(* IEC 61131-3 sources: CodesysTest/export/SX.dev/Plc Logic/Application, 8 files *)

(* ---- Counters.gvl.st ---- *)
(*#-#-#-#-#-#-#-#-#-#---Declaration---#-#-#-#-#-#-#-#-#-#-#-#-#*)

{attribute 'qualified_only'}
VAR_GLOBAL
	jawCycleTestCount : FB_MachineCounter(name := 'Jaw Cycle Test Counter');
	baggerCycles : FB_MachineCounter(name := 'Bagger Cycle Counter');
	pressureBarCycles : FB_MachineCounter(name := 'Pressure Bar Cycle Counter');
	(*Counters*)

	//passthroughChanges : FB_MachineCounter(name := 'Passthrough Changes Counter');
	//loadPlateCycles : FB_MachineCounter(name := 'Load Plate Cycle Counter');
	//printerCycles : FB_MachineCounter(name := 'Printer Cycle Counter');
	//motorizedSealFlattenerCycles : FB_MachineCounter(name := 'Motorized Seal Flattener Cycles');
	//bagOpenRetryTotal : FB_MachineCounter(name := 'Bag Open Retry Totals');
END_VAR

(* ---- Globals.gvl.st ---- *)
(*#-#-#-#-#-#-#-#-#-#---Declaration---#-#-#-#-#-#-#-#-#-#-#-#-#*)

{attribute 'qualified_only'}
{attribute 'global_init_slot' := '49994'}
VAR_GLOBAL
	SystemLog : FB_InternalLogger;

END_VAR

VAR_GLOBAL CONSTANT
	MAX_LOGGED_ITEMS : UINT := 500;	// Max items to be logged
	STEPS_PER_INCH_IBD : DINT := 1250;
	STEPS_PER_INCH_JAW : DINT := 1250;
	STEPS_PER_INCH_LOAD_PLATE : DINT := 931;
	STEPS_PER_INCH_FILM : DINT := 1000;
	SERIAL_BUFFER_SIZE : BYTE := 50;
	SEAL_TO_PHOTOEYE_DISTANCE : REAL := 4.65;
END_VAR

(* ---- PersistentVars.gvl.st ---- *)
(*#-#-#-#-#-#-#-#-#-#---Declaration---#-#-#-#-#-#-#-#-#-#-#-#-#*)

{attribute 'qualified_only'}
VAR_GLOBAL PERSISTENT RETAIN
	// Generated instance path of persistent variable
	HMIData.bagsMade: UDINT;
	// Generated instance path of persistent variable
	HMIData.batchEnable: BOOL;
	// Generated instance path of persistent variable
	HMIData.batchSetting: UDINT := UDINT#10;
	// Generated instance path of persistent variable
	HMIData.batchCount: UDINT;
	// Generated instance path of persistent variable
	HMIData.headCycleCount: UDINT;
	// Generated instance path of persistent variable
	HMIData.pressureBarOpenDelay: REAL;
	// Generated instance path of persistent variable
	HMIData.pressureBarCloseDelay: REAL;
	// Generated instance path of persistent variable
	HMIData.passthroughSetting: REAL := REAL#5.5;
	// Generated instance path of persistent variable
	HMIData.sealBarDwell: REAL := REAL#0.18;
	// Generated instance path of persistent variable
	HMIData.sealBarCool: REAL := REAL#0.25;
	// Generated instance path of persistent variable
	HMIData.bagSkirtLength: REAL := 2.0;
	// Generated instance path of persistent variable
	HMIData.bagLength: REAL := REAL#17.62;
	// Generated instance path of persistent variable
	HMIData.bagWidth: REAL := 11.0;
	// Generated instance path of persistent variable
	HMIData.bagThickness: REAL := REAL#2.5;
	// Generated instance path of persistent variable
	HMIData.bagForwardSpeed: UDINT := UDINT#40;
	// Generated instance path of persistent variable
	HMIData.bagReverseSpeed: UDINT := UDINT#8;
	// Generated instance path of persistent variable
	HMIData.printSpeed: UDINT := UDINT#6;
	// Generated instance path of persistent variable
	HMIData.printLength: REAL := REAL#3;
	// Generated instance path of persistent variable
	HMIData.printOffset: REAL := REAL#8;
	// Generated instance path of persistent variable
	HMIData.fillerCountSetting: UDINT;
	// Generated instance path of persistent variable
	HMIData.fillerCurrentCount: UDINT;
	// Generated instance path of persistent variable
	HMIData.fillerDropTime: REAL;
	// Generated instance path of persistent variable
	HMIData.loadPlateDelay: REAL;
	// Generated instance path of persistent variable
	HMIData.loadPlateDwell: REAL := REAL#0.1;
	// Generated instance path of persistent variable
	HMIData.IBDInUse: BOOL := TRUE;
	// Generated instance path of persistent variable
	HMIData.IBDInstalled: BOOL := TRUE;
	// Generated instance path of persistent variable
	HMIData.IBDOpenMotionProfile: sctMotionProfile := STRUCT(velo := REAL#9, accel := REAL#30, decel := REAL#50, current := REAL#100);
	// Generated instance path of persistent variable
	HMIData.IBDCloseMotionProfile: sctMotionProfile := STRUCT(velo := REAL#15, accel := REAL#10, decel := REAL#10, current := REAL#50);
	// Generated instance path of persistent variable
	HMIData.IBDZeroOffset: REAL := REAL#2;
	// Generated instance path of persistent variable
	HMIData.jawCloseDelay: REAL := REAL#0.1;
	// Generated instance path of persistent variable
	HMIData.jawClosePositionSetting: REAL := REAL#-0.45;
	// Generated instance path of persistent variable
	HMIData.jawOpenMotionProfile: sctMotionProfile := STRUCT(velo := REAL#14, accel := REAL#300, decel := REAL#300, current := REAL#100);
	// Generated instance path of persistent variable
	HMIData.jawCloseMotionProfile: sctMotionProfile := STRUCT(velo := REAL#14, accel := REAL#10, decel := REAL#10, current := REAL#100);
	// Generated instance path of persistent variable
	HMIData.jawCycleTestCycles: DINT;
	// Generated instance path of persistent variable
	HMIData.jawCycleTestActive: BOOL;
	// Generated instance path of persistent variable
	HMIData.jawZeroOffset: REAL := REAL#2;
	// Generated instance path of persistent variable
	HMIData.lastCycleTime: REAL;
	// Generated instance path of persistent variable
	HMIData.bagDropClearanceDwell: REAL := REAL#0.5;
	// Generated instance path of persistent variable
	HMIData.averageCycleTime: REAL;
	// Generated instance path of persistent variable
	HMIData.currentJobID: INT;
	// Generated instance path of persistent variable
	HMIData.separateBeforeSeal: BOOL := TRUE;
	// Generated instance path of persistent variable
	HMIData.partsCounterEnable: BOOL;
	// Generated instance path of persistent variable
	HMIData.partsCounterCount: UDINT;
	// Generated instance path of persistent variable
	HMIData.partsCounterSetting: UDINT;
	// Generated instance path of persistent variable
	HMIData.consecutiveBagsEnable: BOOL;
	// Generated instance path of persistent variable
	HMIData.consecutiveBagsCount: UDINT;
	// Generated instance path of persistent variable
	HMIData.consecutiveBagsSetting: UDINT;
	// Generated instance path of persistent variable
	HMIData.printerInstalled: BOOL := TRUE;
	// Generated instance path of persistent variable
	HMIData.printerInUse: BOOL := TRUE;
	// Generated instance path of persistent variable
	HMIData.printerCancelRequest: BOOL;
	// Generated instance path of persistent variable
	HMIData.barcodeVerifierInstalled: BOOL := TRUE;
	// Generated instance path of persistent variable
	HMIData.barcodeGoodReadCount: UDINT;
	// Generated instance path of persistent variable
	HMIData.barcodeBadReadCount: UDINT;
	// Generated instance path of persistent variable
	HMIData.barcodeBadReadFaultSetting: UDINT;
	// Generated instance path of persistent variable
	HMIData.barcodeStartPosition: REAL;
	// Generated instance path of persistent variable
	HMIData.barcodeScanDistance: REAL := REAL#1;
	// Generated instance path of persistent variable
	HMIData.barcodeVerifierInUse: BOOL := TRUE;
	// Generated instance path of persistent variable
	HMIData.loadPlateInstalled: BOOL := TRUE;
	// Generated instance path of persistent variable
	HMIData.loadPlateLoweredPositionSetting: REAL := 0.0;
	// Generated instance path of persistent variable
	HMIData.loadPlateRaisedPositionSetting: REAL := 1.0;
	// Generated instance path of persistent variable
	HMIData.loadPlateInUse: BOOL := TRUE;
	// Generated instance path of persistent variable
	HMIData.loadPlateRaiseProfile: sctMotionProfile := STRUCT(velo := REAL#3, accel := REAL#100, decel := REAL#10, current := REAL#100);
	// Generated instance path of persistent variable
	HMIData.loadPlateLowerProfile: sctMotionProfile := STRUCT(velo := REAL#5, accel := REAL#100, decel := REAL#100, current := REAL#100);
	// Generated instance path of persistent variable
	HMIData.fillerEnable: BOOL;
	// Generated instance path of persistent variable
	HMIData.autoModeEnable: BOOL;
	// Generated instance path of persistent variable
	HMIData.autoModeDwell: REAL;
	// Generated instance path of persistent variable
	HMIData.dryCycleEnable: BOOL;
END_VAR

(* ---- DeviceChecker.pou.st ---- *)
(*#-#-#-#-#-#-#-#-#-#---Declaration---#-#-#-#-#-#-#-#-#-#-#-#-#*)

FUNCTION_BLOCK DeviceChecker
VAR_INPUT
END_VAR
VAR_OUTPUT
	uiNodes			: UINT;		// number of nodes in device tree
	uiUnknown		: UINT;		// number of devices in unkown state
	uiStopped		: UINT;		// number of devices in stopped state
	uiRunning		: UINT;		// number of devices in running state
	uiError			: UINT;		// number of devices in error state
	uiNotConfigured : UINT;		// number of devices in not configured state
	uiNotFound		: UINT;		// number of devices in not found state
	uiDisabled		: UINT;		// number of disabled devices
END_VAR
VAR
	_itfCurrentNotRunning	: DED.INode;
	_itfNode				: DED.INode;
	_itfDevice				: DED.IDevice;
	_itfBus					: DED.IBus;
END_VAR
(*#-#-#-#-#-#-#-#-#-#---Implementation---#-#-#-#-#-#-#-#-#-#-#-#-#*)

uiNodes			:= 0;
uiUnknown		:= 0;
uiStopped		:= 0;
uiRunning		:= 0;
uiError			:= 0;
uiNotConfigured := 0;
uiNotFound		:= 0;
uiDisabled		:= 0;

// GetRoot() returns INode of the PLC
_itfNode := DED.GetRoot();

REPEAT
	(* cast INode to IDevice *)
	_itfDevice := DED.INode_TO_IDevice(_itfNode);
	(* always check if casting this node was successful!!! *)
	IF _itfDevice <> 0 THEN

		CASE _itfDevice.GetDeviceState() OF
		DED.DEVICE_STATE.UNKNOWN:
			uiUnknown := uiUnknown + 1;
		DED.DEVICE_STATE.STOPPED:
			uiStopped := uiStopped + 1;
		DED.DEVICE_STATE.RUNNING:
			uiRunning := uiRunning + 1;
		DED.DEVICE_STATE.ERROR:
			uiError := uiError + 1;
		DED.DEVICE_STATE.NOT_CONFIGURED:
			uiNotConfigured := uiNotConfigured + 1;
		DED.DEVICE_STATE.NOT_FOUND:
			uiNotFound := uiNotFound + 1;
		DED.DEVICE_STATE.DISABLED:
			uiDisabled := uiDisabled + 1;
		END_CASE

	ELSE
		(* the current node is not an IDevice. Try to cast it to IBus (e.g. CANbus does not implement IDevice, but IBus ) *)
		_itfBus := DED.INode_TO_IBus(_itfNode);
		IF _itfBus <> 0 THEN
			CASE _itfBus.GetBusState() OF
			DED.BUS_STATE.DISABLED:
				uiDisabled := uiDisabled + 1;
			DED.BUS_STATE.ERROR:
				uiError := uiError + 1;
			DED.BUS_STATE.RUNNING:
				uiRunning := uiRunning + 1;
			DED.BUS_STATE.STOPPED:
				uiStopped := uiStopped + 1;
			DED.BUS_STATE.UNKNOWN:
				uiUnknown := uiUnknown + 1;
			END_CASE
		END_IF

	END_IF

	(* total node count *)
	uiNodes := uiNodes + 1;

	(* get the next node from depth-first search*)
	_itfNode := DED.GetNextNode(_itfNode);
UNTIL
	_itfNode = 0
END_REPEAT

(* ---- Devices.pou.st ---- *)
(*#-#-#-#-#-#-#-#-#-#---Declaration---#-#-#-#-#-#-#-#-#-#-#-#-#*)

PROGRAM Devices
VAR

END_VAR
VAR_IN_OUT

END_VAR

VAR_OUTPUT

	pressureBarSolenoidValve : FB_DoubleSolenoidOpenCenterActuator(name := 'Pressure Bar SV');
	sealBarSolenoidValve : FB_SingleSolenoidNormallyRetractedActuator(name := 'Seal Bar SV');
	HPA_LPA_SolenoidValve : FB_DoubleSolenoidClosedCenterActuator(name := 'HPA/LPA SV');
	loadPlateSolenoidValve : FB_DoubleSolenoidOpenCenterActuator(name := 'Load Plate SV');
	bagOpenFingersSolenoidValve : FB_DoubleSolenoidOpenCenterActuator(name := 'BOF SV');
	printHeadSolenoidValve : FB_SingleSolenoidNormallyRetractedActuator(name := 'Print Head SV');
	vacuumSolenoidValve : FB_VacuumGenerator(name := 'Vacuum SV');
	sealFlattenersVertAxisSolenoidValve : FB_DoubleSolenoidOpenCenterActuator(name := 'Seal Flattener Vert SV');
	loadShelfSolenoidValve : FB_DoubleSolenoidOpenCenterActuator(name := 'Load Shelf SV');
	blankSolenoidValve : FB_SolenoidValve(name := 'Blank SV');
	i : UINT;

END_VAR
(*#-#-#-#-#-#-#-#-#-#---Implementation---#-#-#-#-#-#-#-#-#-#-#-#-#*)

(* ---- PLC_PRG.pou.st ---- *)
(*#-#-#-#-#-#-#-#-#-#---Declaration---#-#-#-#-#-#-#-#-#-#-#-#-#*)

PROGRAM PLC_PRG
VAR

	firstScanDone: BOOL;
	cycleStartONS : FB_ONS;
	powerUpFrontJawMotor : Sharp_Motion.MC_Power;
	powerUpRearJawMotor : Sharp_Motion.MC_Power;
	powerUpBothJawMotors : Sharp_Motion.MC_Power;
	powerUpLoadPlateMotor : Sharp_Motion.MC_Power;
	powerUpBagDeliveryMotor : Sharp_Motion.MC_Power;
	powerUpIBDMotor : Sharp_Motion.MC_Power;
	UN00_SXMachine : FB_UN00_SharpMachine(name := 'UN00 - Sharp SX');
	EM01_SXBaggerHead : EM01_BaggerHead(name := 'EM01 - SX Bagger Head');
	EM02_SXDischarge : EM02_Discharge(name := 'EM02 - SX Discharge');
	baggerCM : EM01_Bagger_Control_Modules;
	bannerManager : FB_BannerManager;
	palmButton : FB_BannerPalmButton;
	topCoverLiftedFault : FB_Fault(name := 'Top Cover Lifeted During Cycle');
	amazonBPM : FB_AmazonThroughput();
	printerLabel : FB_PrinterSerial();
	autoModeTimer : Standard.TON;
	autoModeKeepCycling : BOOL;
	autoModeInitiateCycleONS : FB_ONS;
	cycleComplete : FB_ONS;
	hIecTask : RTS_IEC_HANDLE;//Declaration of the variable hIecTask
	teachPhotoeyeTimer : Standard.TOF() := (PT := T#3S);
END_VAR(*#-#-#-#-#-#-#-#-#-#---Implementation---#-#-#-#-#-#-#-#-#-#-#-#-#*)

//	Program: PLC_PRG
//	Description: Base program for the 1179/1181 SX.
//
//	Created by: Ben Hess
//	Created Date:

// Initialze global objects on first scan
IF NOT firstScanDone THEN
	GlobalObjects.CollectionOfInitialzable.InitializeAll();
	GlobalObjects.CollectionOfLoggable.RegisterAll(internalLogger := Globals.SystemLog);
	GlobalObjects.CollectionOfFaults.FaultUpdateForHMI();
	hIecTask := IecTaskGetCurrent(0);
	IecTaskDisableWatchdog(hIecTask); // Watchdog disabled
	firstScanDone := TRUE;
END_IF

// Teach bag photoeye
teachPhotoeyeTimer(IN := HMIData.teachBagPhotoeye, Q => oTeachPhotoeye);
HMIData.teachingBagPhoteye := oTeachPhotoeye;

// Use fault collection for faultActive indication
HMIData.faultActive := GlobalObjects.CollectionOfActiveFaults.faultActive;

// Cycle start conditions
// Auto mode dwell timer
autoModeTimer(PT := TO_TIME(HMIData.autoModeDwell * 1000), IN := autoModeKeepCycling AND UN00_SXMachine.currentState = PACK_ML.State.Execute AND NOT HMIData.inCycle);
// Start from Cycle Start input
cycleStartONS(clk := iCycleStart);
// All start conditions
IF HMIData.initiateCycle OR cycleStartONS.OSR OR autoModeTimer.Q THEN
	IF UN00_SXMachine.currentState = PACK_ML.State.Execute AND NOT HMIData.inCycle THEN
		EM01_SXBaggerHead.StartCycle();
		IF HMIData.autoModeEnable THEN
			autoModeKeepCycling := TRUE;
		END_IF
	END_IF
	HMIData.initiateCycle := FALSE;
END_IF
// Unlatch flag for auto mode when faulted or stopped
IF UN00_SXMachine.currentState <> PACK_ML.State.Execute OR HMIData.ackAllFaults OR NOT HMIData.autoModeEnable THEN
	autoModeKeepCycling := FALSE;
END_IF

// Only faults execute automatically to handle acking and clearing without being run in each FB that contains them
IF firstScanDone THEN
	GlobalObjects.CollectionOfExecutable.ExecuteAll();
END_IF

// Power up all motors
powerUpFrontJawMotor(Enable := TRUE, Axis := baggerCM.jawFrontMotor);
powerUpFrontJawMotor.DriveStart := TRUE;
powerUpFrontJawMotor.RegulatorOn := TRUE;

powerUpRearJawMotor(Enable := TRUE, Axis := baggerCM.jawRearMotor);
powerUpRearJawMotor.DriveStart := TRUE;
powerUpRearJawMotor.RegulatorOn := TRUE;

powerUpBothJawMotors(Enable := TRUE, Axis := baggerCM.jawBothMotors);
powerUpBothJawMotors.DriveStart := TRUE;
powerUpBothJawMotors.RegulatorOn := TRUE;

powerUpLoadPlateMotor(Enable := HMIData.loadPlateInstalled, Axis := baggerCM.loadPlateMotor);
powerUpLoadPlateMotor.DriveStart := HMIData.loadPlateInstalled;
powerUpLoadPlateMotor.RegulatorOn := HMIData.loadPlateInstalled;

powerUpBagDeliveryMotor(Enable := TRUE, Axis := baggerCM.bagDeliveryFrontMotor);
powerUpBagDeliveryMotor.DriveStart := TRUE;
powerUpBagDeliveryMotor.RegulatorOn := TRUE;

powerUpIBDMotor(Enable := HMIData.IBDInstalled, Axis := baggerCM.IBDMotor);
powerUpIBDMotor.DriveStart := HMIData.IBDInstalled;
powerUpIBDMotor.RegulatorOn := HMIData.IBDInstalled;

// Disable Modbus device tree objects if option not installed
IF NOT HMIData.loadPlateInstalled THEN
	Load_Plate_Motor.Enable := FALSE;
ELSE
	Load_Plate_Motor.Enable := TRUE;
END_IF

IF NOT HMIData.IBDInstalled THEN
	IBD_Motor.Enable := FALSE;
ELSE
	IBD_Motor.Enable := TRUE;
END_IF

// Barcode Verifier manual trigger
IF HMIData.barcodeVerifierTrigger THEN
	baggerCM.barcodeVerifier.TriggerImmediate();
	HMIData.barcodeVerifierTrigger := FALSE;
END_IF

// Printer sample label sending
IF HMIData.sendSampleLabels AND NOT printerLabel.xExecute THEN
	printerLabel.xExecute := TRUE;
	printerLabel.sendSampleLabel := TRUE;
	printerLabel.sendClearLabel := FALSE;
	HMIData.sendSampleLabels := FALSE;
ELSIF HMIData.clearAllLabels AND NOT printerLabel.xExecute THEN
	printerLabel.xExecute := TRUE;
	printerLabel.sendSampleLabel := FALSE;
	printerLabel.sendClearLabel := TRUE;
	HMIData.clearAllLabels := FALSE;
END_IF

IF printerLabel.xDone THEN
	printerLabel.xExecute := FALSE;
END_IF
printerLabel();

// Run collection of bagger control modules
baggerCM();

// Set bagger head control modules
EM01_SXBaggerHead(
	bagOpenFingers:= baggerCM.dummyBOF,
	sealFlatteners:= baggerCM.dummySealFlatteners,
	sealer:= baggerCM.sealWire,
	pressureBar:= baggerCM.dualMotorPassthrough,
	printer:= baggerCM.labelPrinter,
	bagDelivery:= baggercm.bagDelivery,
	vacuumBagOpen:= baggerCM.dummyVacuumCups,
	IBD:= baggerCM.IBD,
	loadPlate:= baggerCM.loadPlate,
	barcodeVerifier:= baggerCM.barcodeVerifier,
	bagOpenAssistEnabled:= FALSE,
	bagOpenSensorEnabled:= FALSE,
	cancelPrint := HMIData.printerCancelRequest,
	separateBeforeSealEnabled:= HMIData.separateBeforeSeal,
	bagOpenRetrySetting:= ,
	newJobLoaded:= ,
	vacuumDwell:= ,
	bagOpenRetryCount=> ,
	failedToOpenBag=> );

EM02_SXDischarge();

// Machine unit
UN00_SXMachine(faultActive:= HMIData.faultActive, resetMachine := HMIData.ackAllFaults, homeMachine := HMIData.homeMachine, currentState=> , baggerHead:= EM01_SXBaggerHead, discharge:= EM02_SXDischarge);

// Trigger fault if top cover lifted during cycle
IF HMIData.inCycle AND NOT iTopCoverClosed THEN
	topCoverLiftedFault.Trigger();
END_IF

// Banner palm button has 4 states - off, solid green, 50/50 green/white rotating, and flashing red
palmButton(
	baggerReady:= UN00_SXMachine.currentState = PACK_ML.State.Execute,
	baggerFaulted:= HMIData.faultActive,
	baggerInCycle:= HMIData.inCycle,
	palmState0Output=> oPalmButton0,
	palmState1Output=> oPalmButton1);

//
// HMI Mapping
//

// Send the list of active fault strings to HMI for viewing
HMIData.activeFaults := GlobalObjects.CollectionOfActiveFaults.ObjNames;

HMIData.inCycle := UN00_SXMachine.baggerManager.BaggerAutoMode.baggerCycleActive;
// PackML state to string for HMI
HMIData.currentPackMLState := UN00_SXMachine.baggerManager.BaggerAutoMode.currentBaggerState;

// Banner manager takes care of the Multistate lamp used as a banner on the proface
bannerManager(
	baggerNotReady:= NOT UN00_SXMachine.currentState = PACK_ML.State.Execute,
	baggerReady:= UN00_SXMachine.currentState = PACK_ML.State.Execute AND NOT HMIData.inCycle,
	baggerInCycle:= HMIData.inCycle,
	noBagCoveringEye:= baggerCM.bagDelivery.noBagOverEye.Active,
	bagFailedToSeperate:= baggerCM.bagDelivery.bagFailedToSeparate.Active,
	pbarObstruction:= baggerCM.dualMotorPassthrough.pressureBarObstructed.Active,
	lightCurtainViolation:= ,
	printHeadFTR:= baggerCM.labelPrinter.printHeadFailToRaise.Active,
	printHeadFTL:= baggerCM.labelPrinter.printHeadFailToLower.Active,
	barcodeFault:= EM01_SXBaggerHead.barcodeVerificationFailed.Active,
	tooManyPartsCounted:= ,
	jawFailedToClose:= baggerCM.dualMotorPassthrough.failedToClose.Active,
	jawFailedToHome:= baggerCM.dualMotorPassthrough.failedToHome.Active,
	filmFeedMotionFault:= ,
	jawMotionFault:= baggerCM.dualMotorPassthrough.bothMotorsFault.Active,
	waitingOnPrinter:= UN00_SXMachine.baggerManager.BaggerAutoMode.releaseAndFeedSubState = RELEASE_FEED_STATES.WaitForPrinter,
	waitingOnFiller:= ,
	batchCounterDone:= ,
	jawNotHomed:= NOT baggerCM.dualMotorPassthrough.IsHomed AND NOT HMIData.inCycle,
	cycleBaggerTForFiller:= ,
	machineNotTested:=  HMIData.bagsMade < 1000,
	loadPlateMotorNotHomed:= NOT baggerCM.loadPlate.IsHomed AND baggerCM.loadPlate.OptionActive,
	loadPlateMotorFaulted:= baggerCM.loadPlate.motorFault.Active,
	loadPlateMotorCommF:= baggerCM.loadPlate.motorCommFault.Active,
	topCoverLiftedFault:= topCoverLiftedFault.Active,
	topCoverLiftedWarning:= NOT iTopCoverClosed AND NOT HMIData.inCycle,
	IBDMotorNotHomed:= NOT baggerCM.IBD.IsHomed AND baggerCM.IBD.OptionActive AND NOT HMIData.inCycle,
	IBDMotorFaulted:= baggerCM.IBD.IBDMotorFault.Active,
	IBDMotorCommF:= baggerCM.IBD.IBDMotorCommFault.Active,
	printerRibbonFault := baggerCM.labelPrinter.ribbonFault.Active,
	printerServiceRequired := baggerCM.labelPrinter.serviceRequired.Active,
	jawFailedToOpen:= baggerCM.dualMotorPassthrough.failedToOpen.Active,
	IBDFailedToClose:= ,
	IBDFailedToOpen:= baggerCM.IBD.failedToOpen.Active,
	messageDisplayIndication=> HMIData.bannerMessageIndication);

// Ready indications for bagger control modules
HMIData.printerReady := baggerCM.labelPrinter.Ready;
HMIData.bagDeliveryReady := baggerCM.bagDelivery.Ready;
HMIData.loadPlateReady := baggerCM.loadPlate.Ready;
HMIData.jawReady := baggerCM.dualMotorPassthrough.Ready;
HMIData.bcvReady := baggerCM.barcodeVerifier.Ready;
HMIData.IBDReady := baggerCM.IBD.Ready;

// Motor data to HMI for troubleshooting
HMIData.frontJawMotorData.ActPos := baggerCM.jawFrontMotor.ActPos;
HMIData.frontJawMotorData.CommandedPos := baggerCM.jawFrontMotor.TargetPosDist;
HMIData.frontJawMotorData.CurrentAlarmCode := baggerCM.jawFrontMotor.alarmCode;

HMIData.rearJawMotorData.ActPos := baggerCM.jawRearMotor.ActPos;
HMIData.rearJawMotorData.CommandedPos := baggerCM.jawRearMotor.TargetPosDist;
HMIData.rearJawMotorData.CurrentAlarmCode := baggerCM.jawRearMotor.alarmCode;

HMIData.IBDMotorData.ActPos := baggerCM.IBDMotor.ActPos;
HMIData.IBDMotorData.CommandedPos := baggerCM.IBDMotor.TargetPosDist;
HMIData.IBDMotorData.CurrentAlarmCode := baggerCM.IBDMotor.alarmCode;

HMIData.loadPlateMotorData.ActPos := baggerCM.loadPlateMotor.ActPos;
HMIData.loadPlateMotorData.CommandedPos := baggerCM.loadPlateMotor.TargetPosDist;
HMIData.loadPlateMotorData.CurrentAlarmCode := baggerCM.loadPlateMotor.alarmCode;

HMIData.bagDeliveryMotorData.alarmCode := baggerCM.bagDeliveryFrontMotor.alarmCode;
HMIData.bagDeliveryMotorData.statusCode := baggerCM.bagDeliveryFrontMotor.statusCode;

// Cycle time and bags made counters
HMIData.cycleTime := UN00_SXMachine.baggerManager.BaggerAutoMode.cycleTime;
HMIData.inCycle := UN00_SXMachine.baggerManager.BaggerAutoMode.cycleTimer.IN;
cycleComplete(CLK := UN00_SXMachine.baggerManager.BaggerAutoMode.cycleComplete);
IF cycleComplete.OSR THEN
	HMIData.bagsMade := HMIData.bagsMade + 1;
END_IF

// Printer and Barcode Verifier combination enable/disable
HMIData.printerAndVerifierEnableIndication := HMIData.printerInUse AND HMIData.barcodeVerifierInUse;
IF HMIData.printerAndVerifierEnablePB THEN
	IF HMIData.printerAndVerifierEnableIndication THEN
		HMIData.printerInUse := FALSE;
		HMIData.barcodeVerifierInUse := FALSE;
	ELSE
		HMIData.printerInstalled := TRUE;
		HMIData.barcodeVerifierInstalled := TRUE;
		HMIData.printerInUse := TRUE;
		HMIData.barcodeVerifierInUse := TRUE;
	END_IF
	HMIData.printerAndVerifierEnablePB := FALSE;
END_IF

// Position Indications for service commands
HMIData.jawService.extendedFeedback := baggerCM.dualMotorPassthrough.IsFullyOpen;
HMIData.jawService.retractedFeedback := baggerCM.dualMotorPassthrough.IsFullyClosed;

HMIData.IBDService.extendedFeedback := baggerCM.IBD._isFullyOpen;
HMIData.IBDService.retractedFeedback := NOT baggerCM.IBD._isFullyOpen;

HMIData.printHeadService.extendedFeedback := iPrintHeadLowered;
HMIData.printHeadService.retractedFeedback := NOT iPrintHeadLowered;

// Amazon Bags per minute throughput calculator
amazonBPM(
	inCycle:= HMIData.inCycle,
	runtimeTimeout:= ,
	reset:= HMIData.BPMReset,
	BPM=> HMIData.BPMBagsPerMinute,
	BPMCycles=> HMIData.BPMBagsMade,
	BPMSeconds=> ,
	BPMIndication=> HMIData.BPMActiveTime);

(* ---- POU.pou.st ---- *)
(*#-#-#-#-#-#-#-#-#-#---Declaration---#-#-#-#-#-#-#-#-#-#-#-#-#*)

PROGRAM POU
VAR
	testASCII : FB_ASCII;
END_VAR
(*#-#-#-#-#-#-#-#-#-#---Implementation---#-#-#-#-#-#-#-#-#-#-#-#-#*)

testASCII();

(* ---- SerialComms.pou.st ---- *)
(*#-#-#-#-#-#-#-#-#-#---Declaration---#-#-#-#-#-#-#-#-#-#-#-#-#*)

PROGRAM SerialComms
VAR
	//testASCII : FB_PrinterSerial;
	serial : FB_CrevisSerial();
	fastBagDelivery : FB_SXBagDelivery(name := 'Bag Delivery') := (_optionEnabled := TRUE, _optionInstalled := TRUE);
	fastBagDeliveryFrontMotor : FB_AppliedMotionMotorASCII;
	powerUpBagDeliveryMotor : Sharp_Motion.MC_Power();
END_VAR
(*#-#-#-#-#-#-#-#-#-#---Implementation---#-#-#-#-#-#-#-#-#-#-#-#-#*)

//testASCII();

powerUpBagDeliveryMotor(Enable := TRUE, Axis := fastBagDeliveryFrontMotor);
powerUpBagDeliveryMotor.DriveStart := TRUE;
powerUpBagDeliveryMotor.RegulatorOn := TRUE;

serial(
	xExecute:= ,
	xDone=> ,
	xBusy=> ,
	xError=> ,
	sendData:= ,
	receivedData=> ,
	inputs:= ADR(serialInputs),
	outputs:= ADR(serialOutputs));

fastBagDeliveryFrontMotor(
	AxisState:= ,
	SetOpMode:= ,
	PowerOn:= ,
	DriveEnable:= ,
	AckError:= ,
	StartHoming:= ,
	Halt:= ,
	NewSetPoint:= ,
	MoveAbs:= ,
	MoveAbsTorque:= ,
	MoveRel:= ,
	MoveVelo:= ,
	TargetPosDist:= ,
	TargetVelocity:= ,
	ProfileVelocity:= ,
	ProfileAcceleration:= ,
	ProfileDeceleration:= ,
	ProfileCurrentLimit:= ,
	QuickStopDeceleration:= ,
	DefaultCurrent:= ,
	ActOpMode=> ,
	CommStatus=> ,
	PowerState=> ,
	EnableState=> ,
	Error=> ,
	ActPos=> ,
	ActVelocity=> ,
	SetPointAck=> ,
	TargetReached=> ,
	InVelocity=> ,
	HomingDone=> ,
	modbusAddress:= ,
	stepsPerInchSP:= Globals.STEPS_PER_INCH_FILM,
	zeroOffset:= ,
	jogForwardCMD:= HMIData.jogFilmForward,
	jogReverseCMD:= HMIData.jogFilmReverse,
	asciiHandler:= SerialComms.serial);

fastBagDelivery(
	simulateIO := HMIData.simulateAllIO,
	dryCycleEnable := HMIData.dryCycleEnable,
	_optionActive=> ,
	printer:= PLC_PRG.baggerCM.labelPrinter,
	bagLength:= HMIData.bagLength,
	feedSpeed:= TO_REAL(HMIData.bagForwardSpeed),
	reverseSpeed:= TO_REAL(HMIData.bagReverseSpeed),
	printSpeed:= TO_REAL(HMIData.printSpeed),
	printOffset:= HMIData.printOffset,
	printLength:= HMIData.printLength,
	maxReverseSetpoint:= 4.0,
	sealOffset:= HMIData.bagSkirtLength,
	distanceFromSealBarToBagEdge:= ,
	distanceFromNipToBagEdge:= ,
	bagPresent:= iBagEdgePhotoeye,
	trapezoidalPercent:= ,
	reverseFault=> ,
	bagFailedToSeparate=> ,
	bagDeliveryMotor:= fastBagDeliveryFrontMotor);
